KUKA KRL data list: ps_604c1_o.dat

&ACCESS RVO
&COMMENT Geom C1 Accelo ANTIGO COM O PTO 60-0682
DEFDAT ps_604c1_O
;FOLD EXTERNAL DECLARATIONS;%{PE}%V2.2.2,%MKUKATPBASIS,%CEXT,%VCOMMON,%P
;FOLD BAS EXT;%{PE}%V2.2.2,%MKUKATPBASIS,%CEXT,%VEXT,%P
EXT  BAS (BAS_COMMAND  :IN,REAL  :IN )
DECL INT SUCCESS
;ENDFOLD
;FOLD A10 EXT;%{E}%V2.2.2,%MKUKATPARC,%CEXT,%VEXT,%P
EXT  A10 (A_CMD_T  :IN,A_STRT_T  :IN,A_WELD_T  :IN,A_END_T  :IN,INT  :IN )
;ENDFOLD
;FOLD A20 EXT;%{E}%V2.2.2,%MKUKATPA20,%CEXT,%VEXT,%P
EXT  A20 (INT  :IN,WELD_ST  :IN,WELD_FI  :IN,INT  :IN )
;ENDFOLD
;FOLD GRIPPER EXT;%{E}%V2.2.2,%MKUKATPGRIPPER,%CEXT,%VEXT,%P
EXT  H50 (INT  :IN,INT  :IN,INT  :IN,GRP_TYP  :IN )
;ENDFOLD
;FOLD SPOT EXT;%{E}%V2.2.2,%MKUKATPSPOT,%CEXT,%VEXT,%P
EXT  USERSPOT (S_COMMAND  :IN,SPOT_TYPE  :IN )
;ENDFOLD
;FOLD TOUCHSENSE EXT;%{E}%V2.2.2,%MKUKATPTS,%CEXT,%VEXT,%P
EXT  H70 (INT  :IN,SRCH_TYP_2  :OUT,E6POS  :IN,SRCH_TYP_3  :IN,SRCH_TYP_2  :IN,SRCH_TYP_2  :IN,SRCH_TYP_2  :IN,SRCH_TYP_2  :IN,SRCH_TYP_2  :IN,INT  :IN )
;ENDFOLD
;FOLD USER EXT;%{}%V2.2.2,%MKUKATPUSER,%CEXT,%VEXT,%P
;Make here your modifications
;ENDFOLD
;ENDFOLD

;# ============ START PATH : swp_p13060r4_ltc_geo_c1 =============
DECL BASIS_SUGG_T LAST_BASIS={POINT1[] "p1289                   ",POINT2[] "p1289                   ",CP_PARAMS[] "CPDAT0                  ",PTP_PARAMS[] "PDAT120                 ",CONT[] "C_PTP                   ",CP_VEL[] "2.0                     ",PTP_VEL[] "80                      "}
DECL E6POS Xp1325={x -664.33252,y 791.078308,z 1371.44495,a 63.5197105,b 34.798481,c -89.5357285,s 2,t 42,e1 0.0,e2 0.0,e3 0.0,e4 0.0,e5 0.0,e6 0.0}
DECL FDAT Fp1325={TOOL_NO 1,BASE_NO 2,IPO_FRAME #BASE}
DECL PDAT PPDAT36={VEL 100.0,ACC 80.0,APO_DIST 100.0}
DECL E6POS Xp1326={x 521.072083,y 797.630676,z 1111.98206,a 70.3121872,b -41.000679,c -60.9436798,s 2,t 43,e1 0.0,e2 0.0,e3 0.0,e4 0.0,e5 0.0,e6 0.0}
DECL FDAT Fp1326={TOOL_NO 1,BASE_NO 2,IPO_FRAME #BASE}
DECL PDAT PPDAT37={VEL 100.0,ACC 80.0,APO_DIST 100.0}
DECL E6POS Xswp_60_0806={x 521.875122,y 874.100708,z 1147.64001,a 70.1288834,b -13.9600601,c -67.1750565,s 2,t 43,e1 0.0,e2 0.0,e3 0.0,e4 0.0,e5 0.0,e6 0.0}
DECL FDAT Fswp_60_0806={TOOL_NO 1,BASE_NO 2,IPO_FRAME #BASE}
DECL PDAT PPDAT38={VEL 60.0,ACC 100.0,APO_DIST 100.0}
DECL E6POS Xswp_60_0804={x 502.324188,y 884.674011,z 1112.979,a 68.8673096,b -13.4421701,c -66.8784866,s 2,t 43,e1 0.0,e2 0.0,e3 0.0,e4 0.0,e5 0.0,e6 0.0}
DECL FDAT Fswp_60_0804={TOOL_NO 1,BASE_NO 2,IPO_FRAME #BASE}
DECL PDAT PPDAT39={VEL 60.0,ACC 100.0,APO_DIST 100.0}
DECL E6POS Xp1317={x 490.735687,y 860.807312,z 1094.17395,a 68.8672638,b -13.4404297,c -66.8604965,s 2,t 43,e1 0.0,e2 0.0,e3 0.0,e4 0.0,e5 0.0,e6 0.0}
DECL FDAT Fp1317={TOOL_NO 1,BASE_NO 2,IPO_FRAME #BASE}
DECL PDAT PPDAT40={VEL 100.0,ACC 80.0,APO_DIST 2.0}
DECL E6POS Xswp_60_0802={x 484.975098,y 890.903381,z 1076.27795,a 67.586853,b -12.6261501,c -65.7211609,s 2,t 43,e1 0.0,e2 0.0,e3 0.0,e4 0.0,e5 0.0,e6 0.0}
DECL FDAT Fswp_60_0802={TOOL_NO 1,BASE_NO 2,IPO_FRAME #BASE}
DECL PDAT PPDAT41={VEL 60.0,ACC 100.0,APO_DIST 100.0}
DECL E6POS Xswp_60_0798={x 440.638794,y 899.939026,z 997.353882,a 69.1042633,b -12.6667299,c -63.8055496,s 2,t 43,e1 0.0,e2 0.0,e3 0.0,e4 0.0,e5 0.0,e6 0.0}
DECL FDAT Fswp_60_0798={TOOL_NO 1,BASE_NO 2,IPO_FRAME #BASE}
DECL PDAT PPDAT43={VEL 60.0,ACC 100.0,APO_DIST 100.0}
DECL E6POS Xswp_60_0794={x 411.720093,y 906.200928,z 940.989624,a 56.0326195,b -27.8478603,c -57.9101295,s 2,t 43,e1 0.0,e2 0.0,e3 0.0,e4 0.0,e5 0.0,e6 0.0}
DECL FDAT Fswp_60_0794={TOOL_NO 1,BASE_NO 2,IPO_FRAME #BASE}
DECL PDAT PPDAT44={VEL 60.0,ACC 100.0,APO_DIST 100.0}
DECL E6POS Xp1282={x 421.36319,y 868.844116,z 954.054626,a 67.8700027,b -12.8819599,c -61.6052208,s 2,t 43,e1 0.0,e2 0.0,e3 0.0,e4 0.0,e5 0.0,e6 0.0}
DECL FDAT Fp1282={TOOL_NO 1,BASE_NO 2,IPO_FRAME #BASE}
DECL PDAT PP_OLP77={VEL 100.0,ACC 80.0,APO_DIST 2.0}
DECL E6POS Xp1316={x 390.931885,y 879.709595,z 901.224915,a 69.7426376,b -11.9074697,c -62.0432701,s 2,t 43,e1 0.0,e2 0.0,e3 0.0,e4 0.0,e5 0.0,e6 0.0}
DECL FDAT Fp1316={TOOL_NO 1,BASE_NO 2,IPO_FRAME #BASE}
DECL PDAT PPDAT45={VEL 100.0,ACC 80.0,APO_DIST 2.0}
DECL E6POS Xswp_60_0792={x 384.494293,y 909.690674,z 893.692627,a 69.2772217,b -11.9066601,c -62.0431099,s 2,t 43,e1 0.0,e2 0.0,e3 0.0,e4 0.0,e5 0.0,e6 0.0}
DECL FDAT Fswp_60_0792={TOOL_NO 1,BASE_NO 2,IPO_FRAME #BASE}
DECL PDAT PPDAT46={VEL 60.0,ACC 100.0,APO_DIST 100.0}
DECL E6POS Xswp_60_0790={x 365.862091,y 912.066406,z 854.786499,a 69.2770767,b -11.9079704,c -62.0428696,s 2,t 43,e1 0.0,e2 0.0,e3 0.0,e4 0.0,e5 0.0,e6 0.0}
DECL FDAT Fswp_60_0790={TOOL_NO 1,BASE_NO 2,IPO_FRAME #BASE}
DECL PDAT PPDAT47={VEL 60.0,ACC 100.0,APO_DIST 100.0}
DECL E6POS Xswp_60_0788={x 348.100586,y 915.637085,z 822.080017,a 70.0882492,b -11.90868,c -62.043869,s 2,t 43,e1 0.0,e2 0.0,e3 0.0,e4 0.0,e5 0.0,e6 0.0}
DECL FDAT Fswp_60_0788={TOOL_NO 1,BASE_NO 2,IPO_FRAME #BASE}
DECL PDAT PPDAT48={VEL 60.0,ACC 100.0,APO_DIST 100.0}
DECL E6POS Xp1321={x 342.879211,y 886.523315,z 804.616272,a 70.0854492,b -11.9079905,c -62.0433807,s 2,t 43,e1 0.0,e2 0.0,e3 0.0,e4 0.0,e5 0.0,e6 0.0}
DECL FDAT Fp1321={TOOL_NO 1,BASE_NO 2,IPO_FRAME #BASE}
DECL PDAT PPDAT49={VEL 100.0,ACC 80.0,APO_DIST 100.0}
DECL E6POS Xswp_60_0786={x 328.104187,y 918.011475,z 780.849121,a 70.0851135,b -11.9079599,c -62.0432701,s 2,t 43,e1 0.0,e2 0.0,e3 0.0,e4 0.0,e5 0.0,e6 0.0}
DECL FDAT Fswp_60_0786={TOOL_NO 1,BASE_NO 2,IPO_FRAME #BASE}
DECL PDAT PPDAT50={VEL 60.0,ACC 100.0,APO_DIST 100.0}
DECL E6POS Xp1322={x 308.105713,y 873.905273,z 742.801514,a 70.0945435,b -11.8402796,c -61.8813286,s 2,t 43,e1 0.0,e2 0.0,e3 0.0,e4 0.0,e5 0.0,e6 0.0}
DECL FDAT Fp1322={TOOL_NO 1,BASE_NO 2,IPO_FRAME #BASE}
DECL PDAT PPDAT51={VEL 100.0,ACC 80.0,APO_DIST 100.0}
DECL E6POS Xp1323={x 291.983704,y 899.691284,z 719.056824,a 66.3057632,b -11.9094105,c -62.04282,s 2,t 43,e1 0.0,e2 0.0,e3 0.0,e4 0.0,e5 0.0,e6 0.0}
DECL FDAT Fp1323={TOOL_NO 1,BASE_NO 2,IPO_FRAME #BASE}
DECL PDAT PPDAT52={VEL 100.0,ACC 80.0,APO_DIST 100.0}
DECL E6POS Xswp_60_0782={x 290.686188,y 922.543274,z 711.495789,a 70.4437027,b -2.78368092,c -62.0385704,s 2,t 43,e1 0.0,e2 0.0,e3 0.0,e4 0.0,e5 0.0,e6 0.0}
DECL FDAT Fswp_60_0782={TOOL_NO 1,BASE_NO 2,IPO_FRAME #BASE}
DECL PDAT PPDAT53={VEL 60.0,ACC 100.0,APO_DIST 100.0}
DECL E6POS Xp1327={x 291.983704,y 899.691284,z 719.056824,a 66.3057632,b -11.9094105,c -62.04282,s 2,t 43,e1 0.0,e2 0.0,e3 0.0,e4 0.0,e5 0.0,e6 0.0}
DECL FDAT Fp1327={TOOL_NO 1,BASE_NO 2,IPO_FRAME #BASE}
DECL PDAT PPDAT55={VEL 100.0,ACC 80.0,APO_DIST 100.0}
DECL E6POS Xp1328={x 210.493896,y 889.613708,z 765.286072,a 66.3057632,b -11.9092798,c -62.0429306,s 2,t 43,e1 0.0,e2 0.0,e3 0.0,e4 0.0,e5 0.0,e6 0.0}
DECL FDAT Fp1328={TOOL_NO 1,BASE_NO 2,IPO_FRAME #BASE}
DECL PDAT PPDAT56={VEL 100.0,ACC 80.0,APO_DIST 100.0}
DECL E6POS Xp1310={x 164.661804,y 887.389221,z 681.890686,a 66.3055801,b -11.9089699,c -62.0430717,s 2,t 43,e1 0.0,e2 0.0,e3 0.0,e4 0.0,e5 0.0,e6 0.0}
DECL FDAT Fp1310={TOOL_NO 1,BASE_NO 2,IPO_FRAME #BASE}
DECL PDAT PP_OLP78={VEL 100.0,ACC 80.0,APO_DIST 2.0}
DECL E6POS XP1226={x 493.117493,y 845.016479,z 1088.927,a 67.585083,b -12.6274004,c -65.7208862,s 2,t 43,e1 0.0,e2 0.0,e3 0.0,e4 0.0,e5 0.0,e6 0.0}
DECL FDAT Fp1226={TOOL_NO 1,BASE_NO 2,IPO_FRAME #BASE}
DECL PDAT PPDAT57={VEL 100.0,ACC 80.0,APO_DIST 2.0}
DECL E6POS XP1227={x 411.549896,y 859.407288,z 1119.46997,a 67.5851822,b -12.62745,c -65.7212067,s 2,t 43,e1 0.0,e2 0.0,e3 0.0,e4 0.0,e5 0.0,e6 0.0}
DECL FDAT Fp1227={TOOL_NO 1,BASE_NO 2,IPO_FRAME #BASE}
DECL PDAT PPDAT58={VEL 100.0,ACC 80.0,APO_DIST 2.0}
DECL E6POS XP1228={x 346.094513,y 858.244324,z 1036.22302,a 67.5846024,b -12.62815,c -65.7201996,s 2,t 43,e1 0.0,e2 0.0,e3 0.0,e4 0.0,e5 0.0,e6 0.0}
DECL FDAT Fp1228={TOOL_NO 1,BASE_NO 2,IPO_FRAME #BASE}
DECL PDAT PPDAT59={VEL 100.0,ACC 80.0,APO_DIST 2.0}
DECL E6POS XP1229={x 437.514099,y 862.001526,z 1006.414,a 67.5844574,b -12.6285801,c -65.7204132,s 2,t 43,e1 0.0,e2 0.0,e3 0.0,e4 0.0,e5 0.0,e6 0.0}
DECL FDAT Fp1229={TOOL_NO 1,BASE_NO 2,IPO_FRAME #BASE}
DECL PDAT PPDAT60={VEL 100.0,ACC 80.0,APO_DIST 2.0}
DECL E6POS XP1230={x 426.082001,y 902.281372,z 978.801819,a 56.6241417,b -27.0060902,c -58.1826096,s 2,t 43,e1 0.0,e2 0.0,e3 0.0,e4 0.0,e5 0.0,e6 0.0}
DECL FDAT Fp1230={TOOL_NO 1,BASE_NO 2,IPO_FRAME #BASE}
DECL PDAT PPDAT61={VEL 60.0,ACC 100.0,APO_DIST 100.0}
DECL E6POS XP1231={x 240.077194,y 877.396423,z 627.976318,a 66.3055115,b -11.9088202,c -62.0430908,s 2,t 43,e1 0.0,e2 0.0,e3 0.0,e4 0.0,e5 0.0,e6 0.0}
DECL FDAT Fp1231={TOOL_NO 1,BASE_NO 2,IPO_FRAME #BASE}
DECL PDAT PPDAT62={VEL 100.0,ACC 80.0,APO_DIST 2.0}
DECL E6POS Xswp_60_0779={x 254.889297,y 922.880188,z 628.238098,a 66.2572021,b -11.8889399,c -62.0574913,s 2,t 43,e1 0.0,e2 0.0,e3 0.0,e4 0.0,e5 0.0,e6 0.0}
DECL FDAT Fswp_60_0779={TOOL_NO 1,BASE_NO 2,IPO_FRAME #BASE}
DECL PDAT PPDAT63={VEL 60.0,ACC 100.0,APO_DIST 100.0}
DECL E6POS Xswp_60_0777={x 236.407806,y 925.075928,z 592.145081,a 66.2562866,b -11.88908,c -62.0577812,s 2,t 43,e1 0.0,e2 0.0,e3 0.0,e4 0.0,e5 0.0,e6 0.0}
DECL FDAT Fswp_60_0777={TOOL_NO 1,BASE_NO 2,IPO_FRAME #BASE}
DECL PDAT PPDAT64={VEL 60.0,ACC 100.0,APO_DIST 100.0}
DECL E6POS Xswp_60_0775={x 221.752106,y 925.719177,z 560.701172,a 66.2563171,b -11.8889704,c -62.057579,s 2,t 43,e1 0.0,e2 0.0,e3 0.0,e4 0.0,e5 0.0,e6 0.0}
DECL FDAT Fswp_60_0775={TOOL_NO 1,BASE_NO 2,IPO_FRAME #BASE}
DECL PDAT PPDAT65={VEL 60.0,ACC 100.0,APO_DIST 100.0}
DECL E6POS XSWP_60_0773={x 209.309692,y 919.801697,z 530.876709,a 105.374901,b 36.6266708,c -50.0655708,s 2,t 43,e1 0.0,e2 0.0,e3 0.0,e4 0.0,e5 0.0,e6 0.0}
DECL FDAT FSWP_60_0773={TOOL_NO 1,BASE_NO 2,IPO_FRAME #BASE}
DECL PDAT PPDAT66={VEL 60.0,ACC 100.0,APO_DIST 100.0}
DECL E6POS Xp1232={x 221.027603,y 886.39093,z 553.484314,a 105.373901,b 36.6275291,c -50.0648804,s 2,t 43,e1 0.0,e2 0.0,e3 0.0,e4 0.0,e5 0.0,e6 0.0}
DECL FDAT Fp1232={TOOL_NO 1,BASE_NO 2,IPO_FRAME #BASE}
DECL PDAT PP_OLP79={VEL 100.0,ACC 85.0,APO_DIST 10.0}
DECL E6POS XSWP_60_0199={x 188.246002,y 878.614075,z 524.359192,a 178.943298,b 65.2382202,c 15.5458603,s 2,t 11,e1 0.0,e2 0.0,e3 0.0,e4 0.0,e5 0.0,e6 0.0}
DECL FDAT FSWP_60_0199={TOOL_NO 1,BASE_NO 2,IPO_FRAME #BASE}
DECL PDAT PPDAT67={VEL 60.0,ACC 100.0,APO_DIST 100.0}
DECL E6POS Xswp_60_0193={x 151.356293,y 697.993774,z 525.967285,a 165.181793,b 69.6872635,c -11.9986296,s 2,t 11,e1 0.0,e2 0.0,e3 0.0,e4 0.0,e5 0.0,e6 0.0}
DECL FDAT Fswp_60_0193={TOOL_NO 1,BASE_NO 2,IPO_FRAME #BASE}
DECL PDAT PPDAT68={VEL 60.0,ACC 100.0,APO_DIST 100.0}
DECL E6POS XSWP_60_0185={x 128.729706,y 516.413086,z 526.116272,a 179.998505,b 62.8476906,c 4.22269821,s 2,t 11,e1 0.0,e2 0.0,e3 0.0,e4 0.0,e5 0.0,e6 0.0}
DECL FDAT FSWP_60_0185={TOOL_NO 1,BASE_NO 2,IPO_FRAME #BASE}
DECL PDAT PPDAT69={VEL 60.0,ACC 100.0,APO_DIST 100.0}
DECL E6POS Xswp_60_0167={x 105.679398,y 90.7325363,z 529.405823,a 179.996201,b 62.9335289,c 3.64202189,s 2,t 11,e1 0.0,e2 0.0,e3 0.0,e4 0.0,e5 0.0,e6 0.0}
DECL FDAT Fswp_60_0167={TOOL_NO 1,BASE_NO 2,IPO_FRAME #BASE}
DECL PDAT PPDAT70={VEL 50.0,ACC 100.0,APO_DIST 100.0}
DECL E6POS XSWP_60_0103={x 33.1900482,y 251.159698,z 159.220795,a 62.1840096,b -81.8501129,c -69.2860031,s 2,t 43,e1 0.0,e2 0.0,e3 0.0,e4 0.0,e5 0.0,e6 0.0}
DECL FDAT FSWP_60_0103={TOOL_NO 1,BASE_NO 2,IPO_FRAME #BASE}
DECL PDAT PPDAT71={VEL 60.0,ACC 100.0,APO_DIST 100.0}
DECL E6POS XSWP_60_0115={x 44.7215118,y 454.82019,z 144.828903,a 79.1381836,b -54.5401001,c -83.5403366,s 2,t 43,e1 0.0,e2 0.0,e3 0.0,e4 0.0,e5 0.0,e6 0.0}
DECL FDAT FSWP_60_0115={TOOL_NO 1,BASE_NO 2,IPO_FRAME #BASE}
DECL PDAT PPDAT72={VEL 60.0,ACC 100.0,APO_DIST 100.0}
DECL E6POS XSWP_60_0117={x 68.6262436,y 676.227905,z 159.911697,a -91.5174103,b -65.2435226,c 82.9550323,s 2,t 43,e1 0.0,e2 0.0,e3 0.0,e4 0.0,e5 0.0,e6 0.0}
DECL FDAT FSWP_60_0117={TOOL_NO 1,BASE_NO 2,IPO_FRAME #BASE}
DECL PDAT PPDAT73={VEL 60.0,ACC 100.0,APO_DIST 100.0}
DECL E6POS Xswp_60_0119={x 72.5080414,y 701.424011,z 168.435501,a 37.5202408,b -85.3696365,c -43.231781,s 2,t 43,e1 0.0,e2 0.0,e3 0.0,e4 0.0,e5 0.0,e6 0.0}
DECL FDAT Fswp_60_0119={TOOL_NO 1,BASE_NO 2,IPO_FRAME #BASE}
DECL PDAT PPDAT74={VEL 60.0,ACC 100.0,APO_DIST 100.0}
DECL E6POS Xswp_60_0121={x 77.653183,y 737.572327,z 180.367798,a 1.03197098,b -86.1405792,c -6.64826822,s 2,t 43,e1 0.0,e2 0.0,e3 0.0,e4 0.0,e5 0.0,e6 0.0}
DECL FDAT Fswp_60_0121={TOOL_NO 1,BASE_NO 2,IPO_FRAME #BASE}
DECL PDAT PPDAT75={VEL 60.0,ACC 100.0,APO_DIST 100.0}
DECL E6POS Xswp_60_0123={x 82.5138702,y 771.063721,z 186.748596,a 37.5705719,b -85.3682404,c -43.2823982,s 2,t 43,e1 0.0,e2 0.0,e3 0.0,e4 0.0,e5 0.0,e6 0.0}
DECL FDAT Fswp_60_0123={TOOL_NO 1,BASE_NO 2,IPO_FRAME #BASE}
DECL PDAT PPDAT76={VEL 60.0,ACC 100.0,APO_DIST 100.0}
DECL E6POS XSWP_60_0127={x 98.7325516,y 829.915222,z 199.673401,a 0.00720024109,b -84.8820724,c -10.1827297,s 2,t 43,e1 0.0,e2 0.0,e3 0.0,e4 0.0,e5 0.0,e6 0.0}
DECL FDAT FSWP_60_0127={TOOL_NO 1,BASE_NO 2,IPO_FRAME #BASE}
DECL PDAT PPDAT77={VEL 60.0,ACC 100.0,APO_DIST 100.0}
DECL E6POS XP1233={x 196.427902,y 797.649475,z 561.333618,a 178.940201,b 65.2386322,c 15.5427704,s 2,t 11,e1 0.0,e2 0.0,e3 0.0,e4 0.0,e5 0.0,e6 0.0}
DECL FDAT Fp1233={TOOL_NO 1,BASE_NO 2,IPO_FRAME #BASE}
DECL PDAT PPDAT78={VEL 100.0,ACC 85.0,APO_DIST 10.0}
DECL E6POS XP1234={x 194.426697,y 709.277771,z 585.929626,a 175.884293,b 65.1324463,c 2.56119204,s 2,t 11,e1 0.0,e2 0.0,e3 0.0,e4 0.0,e5 0.0,e6 0.0}
DECL FDAT Fp1234={TOOL_NO 1,BASE_NO 2,IPO_FRAME #BASE}
DECL PDAT PPDAT79={VEL 100.0,ACC 85.0,APO_DIST 10.0}
DECL E6POS XP1235={x 143.495499,y 592.479614,z 531.168823,a 175.481201,b 65.6446304,c -1.18967199,s 2,t 11,e1 0.0,e2 0.0,e3 0.0,e4 0.0,e5 0.0,e6 0.0}
DECL FDAT Fp1235={TOOL_NO 1,BASE_NO 2,IPO_FRAME #BASE}
DECL PDAT PPDAT80={VEL 100.0,ACC 85.0,APO_DIST 10.0}
DECL E6POS XP1236={x 156.862396,y 516.407227,z 580.971191,a 179.998306,b 62.8476715,c 4.22266483,s 2,t 11,e1 0.0,e2 0.0,e3 0.0,e4 0.0,e5 0.0,e6 0.0}
DECL FDAT Fp1236={TOOL_NO 1,BASE_NO 2,IPO_FRAME #BASE}
DECL PDAT PPDAT81={VEL 100.0,ACC 85.0,APO_DIST 10.0}
DECL E6POS XP1237={x 254.760406,y 501.1203,z 792.022827,a 173.335602,b 72.0107269,c -1.42356503,s 2,t 11,e1 0.0,e2 0.0,e3 0.0,e4 0.0,e5 0.0,e6 0.0}
DECL FDAT Fp1237={TOOL_NO 1,BASE_NO 2,IPO_FRAME #BASE}
DECL PDAT PPDAT82={VEL 100.0,ACC 85.0,APO_DIST 10.0}
DECL E6POS XP1238={x 257.313507,y 243.034302,z 797.192383,a 173.344406,b 72.0115509,c -1.41443896,s 2,t 11,e1 0.0,e2 0.0,e3 0.0,e4 0.0,e5 0.0,e6 0.0}
DECL FDAT Fp1238={TOOL_NO 1,BASE_NO 2,IPO_FRAME #BASE}
DECL PDAT PPDAT83={VEL 100.0,ACC 85.0,APO_DIST 10.0}
DECL E6POS XP1239={x 144.798004,y 123.605598,z 592.043274,a 179.228195,b 65.0072174,c 3.1434319,s 2,t 11,e1 0.0,e2 0.0,e3 0.0,e4 0.0,e5 0.0,e6 0.0}
DECL FDAT Fp1239={TOOL_NO 1,BASE_NO 2,IPO_FRAME #BASE}
DECL PDAT PPDAT84={VEL 100.0,ACC 85.0,APO_DIST 10.0}
DECL E6POS XP1240={x 179.080597,y 132.7565,z 671.88739,a 178.561401,b 69.1954422,c 0.682946622,s 2,t 11,e1 0.0,e2 0.0,e3 0.0,e4 0.0,e5 0.0,e6 0.0}
DECL FDAT Fp1240={TOOL_NO 1,BASE_NO 2,IPO_FRAME #BASE}
DECL PDAT PPDAT85={VEL 100.0,ACC 85.0,APO_DIST 10.0}
DECL E6POS XP1241={x -440.210693,y 288.873108,z 705.667175,a 145.069901,b 65.5228577,c -22.6158199,s 2,t 10,e1 0.0,e2 0.0,e3 0.0,e4 0.0,e5 0.0,e6 0.0}
DECL FDAT Fp1241={TOOL_NO 1,BASE_NO 2,IPO_FRAME #BASE}
DECL PDAT PPDAT86={VEL 100.0,ACC 85.0,APO_DIST 10.0}
DECL E6POS XP1242={x -392.090698,y 312.830902,z 86.7444916,a -51.7184601,b -78.2493668,c 42.6988411,s 2,t 42,e1 0.0,e2 0.0,e3 0.0,e4 0.0,e5 0.0,e6 0.0}
DECL FDAT Fp1242={TOOL_NO 1,BASE_NO 2,IPO_FRAME #BASE}
DECL PDAT PPDAT87={VEL 100.0,ACC 85.0,APO_DIST 10.0}
DECL E6POS XP1243={x 41.6715813,y 247.586899,z 121.7099,a 47.1596909,b -83.5169983,c -54.4612617,s 2,t 43,e1 0.0,e2 0.0,e3 0.0,e4 0.0,e5 0.0,e6 0.0}
DECL FDAT Fp1243={TOOL_NO 1,BASE_NO 2,IPO_FRAME #BASE}
DECL PDAT PPDAT88={VEL 100.0,ACC 85.0,APO_DIST 10.0}
DECL E6POS XP1244={x 43.6024094,y 388.292389,z 103.355003,a 47.1433296,b -83.5185623,c -54.4453392,s 2,t 43,e1 0.0,e2 0.0,e3 0.0,e4 0.0,e5 0.0,e6 0.0}
DECL FDAT Fp1244={TOOL_NO 1,BASE_NO 2,IPO_FRAME #BASE}
DECL PDAT PPDAT89={VEL 100.0,ACC 85.0,APO_DIST 10.0}
DECL E6POS XP1245={x 40.8675194,y 246.726395,z 111.085098,a 47.1441689,b -83.5185089,c -54.4452019,s 2,t 43,e1 0.0,e2 0.0,e3 0.0,e4 0.0,e5 0.0,e6 0.0}
DECL FDAT Fp1245={TOOL_NO 1,BASE_NO 2,IPO_FRAME #BASE}
DECL PDAT PPDAT90={VEL 100.0,ACC 85.0,APO_DIST 10.0}
DECL E6POS XP1246={x 43.6024094,y 388.292389,z 103.355003,a 47.1433296,b -83.5185623,c -54.4453392,s 2,t 43,e1 0.0,e2 0.0,e3 0.0,e4 0.0,e5 0.0,e6 0.0}
DECL FDAT Fp1246={TOOL_NO 1,BASE_NO 2,IPO_FRAME #BASE}
DECL PDAT PPDAT91={VEL 100.0,ACC 85.0,APO_DIST 10.0}
DECL E6POS XP1247={x -387.1185,y 444.809814,z 131.930099,a 47.1437798,b -83.5184402,c -54.4458389,s 2,t 42,e1 0.0,e2 0.0,e3 0.0,e4 0.0,e5 0.0,e6 0.0}
DECL FDAT Fp1247={TOOL_NO 1,BASE_NO 2,IPO_FRAME #BASE}
DECL PDAT PPDAT92={VEL 100.0,ACC 85.0,APO_DIST 10.0}
DECL E6POS XP1248={x -352.059601,y 725.168518,z 105.862503,a 47.1415901,b -83.518158,c -54.4438095,s 2,t 42,e1 0.0,e2 0.0,e3 0.0,e4 0.0,e5 0.0,e6 0.0}
DECL FDAT Fp1248={TOOL_NO 1,BASE_NO 2,IPO_FRAME #BASE}
DECL PDAT PPDAT93={VEL 100.0,ACC 85.0,APO_DIST 10.0}
DECL E6POS XP1249={x 65.9035492,y 679.190002,z 102.245201,a -88.8125305,b -70.7309723,c 80.429657,s 2,t 43,e1 0.0,e2 0.0,e3 0.0,e4 0.0,e5 0.0,e6 0.0}
DECL FDAT Fp1249={TOOL_NO 1,BASE_NO 2,IPO_FRAME #BASE}
DECL PDAT PPDAT94={VEL 100.0,ACC 85.0,APO_DIST 10.0}
DECL E6POS Xswp_60_0125={x 92.3916016,y 801.691772,z 195.440704,a 37.5680008,b -85.3693314,c -43.2796211,s 2,t 43,e1 0.0,e2 0.0,e3 0.0,e4 0.0,e5 0.0,e6 0.0}
DECL FDAT Fswp_60_0125={TOOL_NO 1,BASE_NO 2,IPO_FRAME #BASE}
DECL PDAT PPDAT95={VEL 60.0,ACC 100.0,APO_DIST 100.0}
DECL E6POS XP1250={x 91.2592163,y 811.730286,z 137.247101,a -3.35188389,b -82.4603882,c -7.55397987,s 2,t 43,e1 0.0,e2 0.0,e3 0.0,e4 0.0,e5 0.0,e6 0.0}
DECL FDAT Fp1250={TOOL_NO 1,BASE_NO 2,IPO_FRAME #BASE}
DECL PDAT PPDAT96={VEL 100.0,ACC 85.0,APO_DIST 10.0}
DECL E6POS XP1251={x -323.091797,y 892.059387,z 192.601501,a -3.35227489,b -82.4598312,c -7.55339193,s 2,t 42,e1 0.0,e2 0.0,e3 0.0,e4 0.0,e5 0.0,e6 0.0}
DECL FDAT Fp1251={TOOL_NO 1,BASE_NO 2,IPO_FRAME #BASE}
DECL PDAT PPDAT97={VEL 100.0,ACC 85.0,APO_DIST 10.0}
DECL E6POS XP1252={x -715.440613,y 852.356384,z 113.869698,a 28.8778992,b -70.7833023,c -37.8725014,s 2,t 42,e1 0.0,e2 0.0,e3 0.0,e4 0.0,e5 0.0,e6 0.0}
DECL FDAT Fp1252={TOOL_NO 1,BASE_NO 2,IPO_FRAME #BASE}
DECL PDAT PPDAT98={VEL 100.0,ACC 85.0,APO_DIST 10.0}
DECL E6POS Xp1253={x -1602.77795,y 2108.78491,z 3027.12598,a -9.24487019,b -6.84731388,c 154.184204,s 2,t 10,e1 0.0,e2 0.0,e3 0.0,e4 0.0,e5 0.0,e6 0.0}
DECL FDAT Fp1253={TOOL_NO 1,BASE_NO 2,IPO_FRAME #BASE}
DECL PDAT PP_OLP80={VEL 100.0,ACC 80.0,APO_DIST 100.0}
DECL E6POS Xp1254={x -1716.86401,y 2155.08789,z 2827.3999,a 97.3066635,b -6.4081521,c 140.431305,s 2,t 11,e1 0.0,e2 0.0,e3 0.0,e4 0.0,e5 0.0,e6 0.0}
DECL FDAT Fp1254={TOOL_NO 1,BASE_NO 2,IPO_FRAME #BASE}
DECL PDAT PP_OLP81={VEL 100.0,ACC 80.0,APO_DIST 100.0}
DECL E6POS Xp1255={x -8.43376446,y 2216.13306,z 2516.70508,a 92.5815735,b -35.877079,c -165.342804,s 2,t 11,e1 0.0,e2 0.0,e3 0.0,e4 0.0,e5 0.0,e6 0.0}
DECL FDAT Fp1255={TOOL_NO 1,BASE_NO 2,IPO_FRAME #BASE}
DECL PDAT PP_OLP82={VEL 100.0,ACC 80.0,APO_DIST 100.0}
DECL E6POS Xp1256={x 652.68042,y 2003.56799,z 472.057709,a 31.7797699,b -21.2542,c -93.9522629,s 2,t 11,e1 0.0,e2 0.0,e3 0.0,e4 0.0,e5 0.0,e6 0.0}
DECL FDAT Fp1256={TOOL_NO 1,BASE_NO 2,IPO_FRAME #BASE}
DECL PDAT PP_OLP83={VEL 100.0,ACC 80.0,APO_DIST 100.0}
DECL E6POS Xp1266={x 998.502319,y 1273.64905,z 66.5208435,a 15.0024405,b 23.3846302,c -82.88134,s 2,t 11,e1 0.0,e2 0.0,e3 0.0,e4 0.0,e5 0.0,e6 0.0}
DECL FDAT Fp1266={TOOL_NO 1,BASE_NO 2,IPO_FRAME #BASE}
DECL PDAT PP_OLP92={VEL 100.0,ACC 85.0,APO_DIST 100.0}
DECL E6POS Xp1267={x 905.289429,y 894.510498,z 56.6472702,a -151.945007,b 76.1717834,c 114.983902,s 2,t 11,e1 0.0,e2 0.0,e3 0.0,e4 0.0,e5 0.0,e6 0.0}
DECL FDAT Fp1267={TOOL_NO 1,BASE_NO 2,IPO_FRAME #BASE}
DECL PDAT PP_OLP93={VEL 100.0,ACC 85.0,APO_DIST 100.0}
DECL E6POS XSWP_60_0629={x 902.09082,y 898.379089,z 17.1980801,a -165.138504,b 69.8017273,c 102.067398,s 2,t 11,e1 0.0,e2 0.0,e3 0.0,e4 0.0,e5 0.0,e6 0.0}
DECL FDAT FSWP_60_0629={TOOL_NO 1,BASE_NO 2,IPO_FRAME #BASE}
DECL PDAT PPDAT102={VEL 60.0,ACC 100.0,APO_DIST 100.0}
DECL E6POS Xp1268={x 905.244385,y 894.501099,z 56.5458183,a -168.025696,b 77.0875015,c 99.3153381,s 2,t 11,e1 0.0,e2 0.0,e3 0.0,e4 0.0,e5 0.0,e6 0.0}
DECL FDAT Fp1268={TOOL_NO 1,BASE_NO 2,IPO_FRAME #BASE}
DECL PDAT PP_OLP94={VEL 100.0,ACC 85.0,APO_DIST 1.0}
DECL E6POS Xp1269={x 1059.79297,y 1435.21399,z 45.848999,a -166.120605,b 68.169693,c 89.2002335,s 2,t 11,e1 0.0,e2 0.0,e3 0.0,e4 0.0,e5 0.0,e6 0.0}
DECL FDAT Fp1269={TOOL_NO 1,BASE_NO 2,IPO_FRAME #BASE}
DECL PDAT PP_OLP95={VEL 100.0,ACC 85.0,APO_DIST 100.0}
DECL E6POS Xp1270={x 697.592529,y 1645.56995,z 200.156296,a 118.7211,b 58.5307884,c 1.76357198,s 2,t 11,e1 0.0,e2 0.0,e3 0.0,e4 0.0,e5 0.0,e6 0.0}
DECL FDAT Fp1270={TOOL_NO 1,BASE_NO 2,IPO_FRAME #BASE}
DECL PDAT PPDAT103={VEL 100.0,ACC 80.0,APO_DIST 30.0}
DECL E6POS Xp1271={x 919.311096,y 2499.61401,z 1179.43799,a -33.1881104,b -86.0368195,c 16.99757,s 2,t 11,e1 0.0,e2 0.0,e3 0.0,e4 0.0,e5 0.0,e6 0.0}
DECL FDAT Fp1271={TOOL_NO 1,BASE_NO 2,IPO_FRAME #BASE}
DECL PDAT PP_OLP96={VEL 100.0,ACC 85.0,APO_DIST 100.0}
DECL E6POS Xp1272={x -47.2550011,y 2196.72192,z 2516.74805,a 140.473602,b -35.9211998,c 165.465393,s 2,t 11}
DECL FDAT Fp1272={TOOL_NO 1,BASE_NO 2,IPO_FRAME #BASE}
DECL PDAT PP_OLP97={VEL 100.0,ACC 85.0,APO_DIST 100.0}
DECL E6POS Xp1273={x -1716.85498,y 2155.09106,z 2827.40405,a 97.3054962,b -6.40859985,c 140.431702,s 2,t 11}
DECL FDAT Fp1273={TOOL_NO 1,BASE_NO 2,IPO_FRAME #BASE}
DECL PDAT PP_OLP98={VEL 100.0,ACC 85.0,APO_DIST 2.0}
DECL E6POS XP1275={x -718.189819,y 623.507874,z 1276.36694,a 67.2133636,b -4.25199986,c -101.8592,s 2,t 42,e1 0.0,e2 0.0,e3 0.0,e4 0.0,e5 0.0,e6 0.0}
DECL FDAT Fp1275={TOOL_NO 1,BASE_NO 2,IPO_FRAME #BASE}
DECL PDAT PPDAT104={VEL 100.0,ACC 80.0,APO_DIST 100.0}
DECL E6POS XP1286={x 207.319901,y 887.483826,z 556.34729,a 176.678497,b 66.9554672,c 13.1319199,s 2,t 11,e1 0.0,e2 0.0,e3 0.0,e4 0.0,e5 0.0,e6 0.0}
DECL FDAT Fp1286={TOOL_NO 1,BASE_NO 2,IPO_FRAME #BASE}
DECL PDAT PPDAT116={VEL 100.0,ACC 80.0,APO_DIST 100.0}
DECL E6POS XSWP_60_0785={x 311.363098,y 918.467285,z 742.579285,a 73.7493896,b 8.35336208,c -63.4957504,s 2,t 43,e1 0.0,e2 0.0,e3 0.0,e4 0.0,e5 0.0,e6 0.0}
DECL FDAT FSWP_60_0785={TOOL_NO 1,BASE_NO 2,IPO_FRAME #BASE}
DECL PDAT PPDAT117={VEL 60.0,ACC 100.0,APO_DIST 100.0}
DECL E6POS XP1287={x -1727.724,y 741.768616,z 413.36261,a 53.5088501,b 25.8493195,c -42.8503609,s 2,t 42,e1 0.0,e2 0.0,e3 0.0,e4 0.0,e5 0.0,e6 0.0}
DECL FDAT Fp1287={TOOL_NO 1,BASE_NO 2,IPO_FRAME #BASE}
DECL PDAT PPDAT118={VEL 100.0,ACC 80.0,APO_DIST 100.0}
DECL E6POS XP1288={x 989.267883,y 1898.39099,z 159.818893,a 30.5781898,b -5.54970407,c -83.0655899,s 2,t 11,e1 0.0,e2 0.0,e3 0.0,e4 0.0,e5 0.0,e6 0.0}
DECL FDAT Fp1288={TOOL_NO 1,BASE_NO 2,IPO_FRAME #BASE}
DECL PDAT PPDAT119={VEL 100.0,ACC 80.0,APO_DIST 100.0}
DECL E6POS Xp1290={x -1470.43396,y 2363.67212,z 2902.18604,a -17.1727791,b -7.94201279,c 145.377304,s 2,t 10,e1 0.0,e2 0.0,e3 0.0,e4 0.0,e5 0.0,e6 0.0}
DECL FDAT Fp1290={TOOL_NO 1,BASE_NO 2,IPO_FRAME #BASE}
DECL PDAT PP_OLP100={VEL 100.0,ACC 80.0,APO_DIST 100.0}
DECL E6POS Xp1291={x -664.33252,y 791.078308,z 1371.44495,a 63.5197105,b 34.798481,c -89.5357285,s 2,t 42,e1 0.0,e2 0.0,e3 0.0,e4 0.0,e5 0.0,e6 0.0}
DECL FDAT Fp1291={TOOL_NO 1,BASE_NO 2,IPO_FRAME #BASE}
DECL PDAT PPDAT121={VEL 100.0,ACC 80.0,APO_DIST 100.0}
DECL E6POS Xp1292={x 528.857422,y 819.397217,z 1132.078,a 79.3153763,b -25.89147,c -65.956337,s 2,t 43,e1 0.0,e2 0.0,e3 0.0,e4 0.0,e5 0.0,e6 0.0}
DECL FDAT Fp1292={TOOL_NO 1,BASE_NO 2,IPO_FRAME #BASE}
DECL PDAT PPDAT122={VEL 100.0,ACC 80.0,APO_DIST 100.0}
DECL E6POS Xp1293={x 486.596497,y 865.466675,z 1088.86804,a 73.0518112,b -19.1729794,c -63.9295502,s 2,t 43,e1 0.0,e2 0.0,e3 0.0,e4 0.0,e5 0.0,e6 0.0}
DECL FDAT Fp1293={TOOL_NO 1,BASE_NO 2,IPO_FRAME #BASE}
DECL PDAT PPDAT123={VEL 100.0,ACC 80.0,APO_DIST 100.0}
DECL E6POS Xswp_60_0803={x 459.463989,y 894.398926,z 1036.474,a 69.1045609,b -12.6666403,c -63.8053284,s 2,t 43,e1 0.0,e2 0.0,e3 0.0,e4 0.0,e5 0.0,e6 0.0}
DECL FDAT Fswp_60_0803={TOOL_NO 1,BASE_NO 2,IPO_FRAME #BASE}
DECL PDAT PPDAT124={VEL 60.0,ACC 100.0,APO_DIST 100.0}
DECL E6POS Xp1294={x 439.661407,y 839.448303,z 1022.94397,a 69.1042175,b -12.66675,c -63.8056297,s 2,t 43,e1 0.0,e2 0.0,e3 0.0,e4 0.0,e5 0.0,e6 0.0}
DECL FDAT Fp1294={TOOL_NO 1,BASE_NO 2,IPO_FRAME #BASE}
DECL PDAT PPDAT125={VEL 100.0,ACC 80.0,APO_DIST 100.0}
DECL E6POS Xp1295={x 275.033203,y 911.768372,z 680.668579,a 66.2555084,b -11.8890104,c -62.0573387,s 2,t 43,e1 0.0,e2 0.0,e3 0.0,e4 0.0,e5 0.0,e6 0.0}
DECL FDAT Fp1295={TOOL_NO 1,BASE_NO 2,IPO_FRAME #BASE}
DECL PDAT PPDAT126={VEL 100.0,ACC 80.0,APO_DIST 100.0}
DECL E6POS Xswp_60_0783={x 279.882385,y 922.796082,z 683.200012,a 66.2555466,b -11.88908,c -62.0570602,s 2,t 43,e1 0.0,e2 0.0,e3 0.0,e4 0.0,e5 0.0,e6 0.0}
DECL FDAT Fswp_60_0783={TOOL_NO 1,BASE_NO 2,IPO_FRAME #BASE}
DECL PDAT PPDAT127={VEL 60.0,ACC 100.0,APO_DIST 100.0}
DECL E6POS Xp1296={x 260.493011,y 878.723206,z 673.048523,a 66.2550812,b -11.8894901,c -62.0564995,s 2,t 43,e1 0.0,e2 0.0,e3 0.0,e4 0.0,e5 0.0,e6 0.0}
DECL FDAT Fp1296={TOOL_NO 1,BASE_NO 2,IPO_FRAME #BASE}
DECL PDAT PPDAT128={VEL 100.0,ACC 80.0,APO_DIST 100.0}
DECL E6POS Xp1304={x -194.8405,y 697.135925,z 794.950623,a 56.4149208,b -12.0441198,c -62.1975899,s 2,t 43,e1 0.0,e2 0.0,e3 0.0,e4 0.0,e5 0.0,e6 0.0}
DECL FDAT Fp1304={TOOL_NO 1,BASE_NO 2,IPO_FRAME #BASE}
DECL PDAT PPDAT129={VEL 100.0,ACC 80.0,APO_DIST 100.0}
DECL E6POS Xp1305={x -1002.54102,y 666.742188,z 501.097198,a 32.1180992,b -6.09636402,c -41.9310112,s 2,t 42,e1 0.0,e2 0.0,e3 0.0,e4 0.0,e5 0.0,e6 0.0}
DECL FDAT Fp1305={TOOL_NO 1,BASE_NO 2,IPO_FRAME #BASE}
DECL PDAT PPDAT130={VEL 100.0,ACC 80.0,APO_DIST 100.0}
DECL E6POS Xp1306={x -3990.21704,y 1999.29895,z 439.963013,a -67.8712234,b 20.1257992,c -45.8926201,s 2,t 34,e1 0.0,e2 0.0,e3 0.0,e4 0.0,e5 0.0,e6 0.0}
DECL FDAT Fp1306={TOOL_NO 1,BASE_NO 2,IPO_FRAME #BASE}
DECL PDAT PPDAT131={VEL 100.0,ACC 80.0,APO_DIST 100.0}
DECL E6POS XP1307={x -2213.3999,y 714.784424,z 649.619202,a -14.9919996,b -6.69824886,c -45.92313,s 2,t 42,e1 0.0,e2 0.0,e3 0.0,e4 0.0,e5 0.0,e6 0.0}
DECL FDAT Fp1307={TOOL_NO 1,BASE_NO 2,IPO_FRAME #BASE}
DECL PDAT PPDAT132={VEL 100.0,ACC 85.0,APO_DIST 2.0}
ENDDAT
